FUNCTION StringBeginsWithAny : BOOL
VAR_INPUT
	text : ANY;
	startsWithString : T_MaxString;
END_VAR
VAR
	textLength : DINT;
	length : DINT;
END_VAR

textLength := TO_DINT(LEN2(text.pValue));
length := LEN(startsWithString);

IF (textLength < length) THEN
	RETURN;
END_IF

StringBeginsWithAny := MEMCMP(pBuf1 := text.pValue, pBuf2 := ADR(startsWithString), n := TO_UDINT(length)) = 0;

END_FUNCTION

(* stored: Version 1.1.0.1
   POU StringBeginsWithAny: Id {80260d38-3b40-4b96-b755-073edaa4e021}, SpecialFunc None *)
